FUNCTION_BLOCK FB_CalcFocalLength2LensSets EXTENDS FB_Fallible IMPLEMENTS I_CalcFocalLength2LensSets
VAR
    iConvertUnits : I_ConvertUnitsLREAL;
    iLensSetCompounder : I_LensSetCompounder;
    iCalcFocalLengthLensSet : I_CalcFocalLengthLensSet;

    {attribute 'pytmc' := 'pv: FocalLength'}
    fbFocalLength : FB_QuantityLREALPublic(Units := 'm');
END_VAR


METHOD Calculate : LREAL
VAR_INPUT
    iSourceDistance : I_QuantityLREAL; // Distance from source to downstream lens.
    iDistanceBetween : I_QuantityLREAL; // Distance between the two lens sets.
    iLensSetUpstream : I_LensSet;
    iLensSetDownstream : I_LensSet;
END_VAR
VAR
    fFocalLengthUpstream : LREAL;
    fFocalLengthDownstream : LREAL;
    fbSourceDistance : FB_QuantityLREALPublic(Units := 'm');
    fbDistanceBetween : FB_QuantityLREALPublic(Units := 'm');
    fFocalLengthCompounded : LREAL;
END_VAR

ClearError();

fFocalLengthUpstream := iCalcFocalLengthLensSet.Calculate(iLensSet := iLensSetUpstream);

IF iCalcFocalLengthLensSet.GetError() THEN
    SetError(Msg :=
        CONCAT('Error returned when attempting to calculate the focal length of the upstream lens set: ',
        iCalcFocalLengthLensSet.GetErrorMsg())
    );
    RETURN;
END_IF

fFocalLengthDownstream := iCalcFocalLengthLensSet.Calculate(iLensSet := iLensSetDownstream);

IF iCalcFocalLengthLensSet.GetError() THEN
    SetError(Msg :=
        CONCAT('Error returned when attempting to calculate the focal length of the downstream lens set: ',
        iCalcFocalLengthLensSet.GetErrorMsg())
    );
    RETURN;
END_IF

iLensSetCompounder.Reset();

iConvertUnits.ConvertQuantityLREAL(
    QuantityToConvert := iSourceDistance,
    DesiredUnits := fbFocalLength.Units,
    ConvertedQuantity => fbSourceDistance
);

IF iConvertUnits.GetError() THEN
    SetError(Msg :=
        CONCAT('Error returned when attempting to convert units of source distance input: ',
        iConvertUnits.GetErrorMsg())
    );
    RETURN;
END_IF

iConvertUnits.ConvertQuantityLREAL(
    QuantityToConvert := iDistanceBetween,
    DesiredUnits := fbFocalLength.Units,
    ConvertedQuantity => fbDistanceBetween
);

IF iConvertUnits.GetError() THEN
    SetError(Msg :=
        CONCAT('Error returned when attempting to convert units of distance between input: ',
        iConvertUnits.GetErrorMsg())
    );
    RETURN;
END_IF


fFocalLengthCompounded := iLensSetCompounder.Compound(
    fFocalLength := fFocalLengthUpstream,
    fSourceDistance := iSourceDistance.Val - iDistanceBetween.Val
);

IF iLensSetCompounder.GetError() THEN
    SetError(Msg :=
        CONCAT('Error returned when attempting to compound the focal length of the upstream lens set: ',
        iLensSetCompounder.GetErrorMsg())
    );
    RETURN;
END_IF

fFocalLengthCompounded := iLensSetCompounder.Compound(
    fFocalLength := fFocalLengthDownstream,
    fSourceDistance := iSourceDistance.Val
);

IF iLensSetCompounder.GetError() THEN
    SetError(Msg :=
        CONCAT('Error returned when attempting to compound the focal length of the downstream lens set: ',
        iLensSetCompounder.GetErrorMsg())
    );
    RETURN;
END_IF

fbFocalLength.Val := fFocalLengthCompounded;

Calculate := fbFocalLength.Val;
END_METHOD


METHOD PROTECTED ClearError

SUPER^.ClearError();

fbFocalLength.ClearError();
END_METHOD


METHOD FB_Init: BOOL
VAR_INPUT
    bInitRetains: BOOL; // TRUE: the retain variables are initialized (reset warm / reset cold)
    bInCopyCode: BOOL;  // TRUE: the instance will be copied to the copy code afterward (online change)

    iConvertUnits : I_ConvertUnitsLREAL;
    iLensSetCompounder : I_LensSetCompounder;
    iCalcFocalLengthLensSet : I_CalcFocalLengthLensSet;
END_VAR

THIS^.iConvertUnits := iConvertUnits;
THIS^.iLensSetCompounder := iLensSetCompounder;
THIS^.iCalcFocalLengthLensSet := iCalcFocalLengthLensSet;
END_METHOD


METHOD PROTECTED SetError
VAR_INPUT
    Msg : T_MaxString;
END_VAR

SUPER^.SetError(Msg := Msg);

fbFocalLength.SetError(Msg := Msg);
END_METHOD

END_FUNCTION_BLOCK

(* stored: Version 1.1.0.1
   POU FB_CalcFocalLength2LensSets: Id {765016df-8fcb-4824-a16c-775f522a9b6b}, SpecialFunc None
   Method Calculate: Id {7fb9b932-86ed-4807-9dba-f0f190f19c1a}
   Method ClearError: Id {344e06d0-6482-4e19-8900-d5c02036c81c}
   Method FB_Init: Id {b6c80088-2bb6-423b-86e6-b931e94ef36c}
   Method SetError: Id {8ac67ccb-16d7-474d-8982-b2e646a3254c} *)
